Staubli VAL3: Axis7Action.pgx

public program Axis7Action(num x_nType (dimensions=1))
begin

  //七轴的IO动作

  switch x_nType

    //点动正
    case 1
      if dDio["O4_b7StopMotor"]==true
        dDio["O4_b7StopMotor"]=false
        delay(0.05)
      endIf
      dDio["O4_b7MoveDir"]=true
      // aioSet(aAio["O4_a7JogVelo"],50)
      delay(0.2)

    break


    //点动负
    case 2
      if dDio["O4_b7StopMotor"]==true
        dDio["O4_b7StopMotor"]=false
        delay(0.05)
      endIf

      dDio["O4_b7MoveDirM"]=true
      //  aioSet(aAio["O4_a7JogVelo"],50)
      delay(0.2)
    break

    //回到机械零位
    case 4
      dDio["O4_b7StopMotor"]=false
      dDio["O4_b7AxisHome"]=true
      delay(0.2)
    break





    //停止运动
    case 6
      dDio["O4_b7StopMotor"]=true
      delay(0.2)
      dDio["O4_b7StopMotor"]=false
    break




    //没有按钮按下
    case 9
      dDio["O4_b7ResetError"]=false
      dDio["O4_b7AxisHome"]=false
      dDio["O4_b7MoveDirM"]=false
      dDio["O4_b7MoveDir"]=false
    break


    //复位
    case 10
      dDio["O4_b7StopMotor"]=false
      dDio["O4_b7ResetError"]=true
      delay(0.2)
      // dDio["O4_b7ResetError"]=false
    break
    default
    break

  endSwitch


end
